// TIA Portal V19 export
DATA_BLOCK "HmiInterface"   // DB164
// stored: MemoryReserve 100, Namespace Unit.Em2
   VAR
      em : "LAF_typeEmInterface";
      jobs : "LAF_typeJobsInterface";   // Interface to control jobs of the EM from an HMI
      sequence : "LAF_typeSequenceInterface";
   END_VAR
BEGIN
END_DATA_BLOCK
